INTERFACE I_CylinderCommand EXTENDS I_Base

METHOD Extend
END_METHOD

METHOD Retract
END_METHOD

END_INTERFACE

(* stored: Version 1.1.0.1, ProductVersion 3.1.4026.18
   Itf I_CylinderCommand: Id {9316dbdd-4257-4531-8caa-9a29fca32a93}
   Method Extend: Id {dba1c55e-e128-498f-a7a4-c0be8e1eb1eb}
   Method Retract: Id {0b64a85a-afac-44ef-89ba-e9a2b4f1fb94} *)
